TYPE InfoDataAdsAddrStateBase_1916E49F :
STRUCT
END_STRUCT
END_TYPE

(* stored: Version 1.2.0.0, ProductVersion 3.1.4024.9
   DUT InfoDataAdsAddrStateBase_1916E49F: Id {0bbc5fa0-9042-4c78-86f8-8f04fa771eeb} *)
